(*
/*
 *****************************************************************************
 * timeUTCToJD: convert struct ccsTIMEVAL into Julian date
 *
 *  IN   ut: time in UT
 *  OUT    : Julian date  
 ***************************************************************************** 
 */
*)
FUNCTION F_timeUTCToJD : LREAL
VAR_INPUT
	ut:	T_TIMEVAL;
END_VAR
VAR
	temp1:	LREAL;
END_VAR

(*
DOUBLE timeUTCToJD(vltTIMEVAL *ut)    /* time in UT                       */
    {
    DOUBLE jd;
    
   /*
    * CONST4 = jd(70-01-01 00:00:00.000000)
    */
    jd = CONST4 + (ut->tv_sec + ut->tv_usec/1000000.)/86400.;
    return(jd);
    }
*)

//F_timeUTCToJD := GCL.C_CONST4 + (UDINT_TO_REAL(ut.tv_sec) + DINT_TO_REAL(ut.tv_usec)/1000000.0)/86400.0;

temp1	:= DINT_TO_LREAL(ut.tv_usec)/1000000.0;
temp1	:= temp1 + UDINT_TO_LREAL(ut.tv_sec);

F_timeUTCToJD := GCL.C_CONST4 + (temp1)/86400.0;

END_FUNCTION

(* stored: Version 1.1.0.1, ProductVersion 3.1.4024.10
   POU F_timeUTCToJD: Id {0fe20a4c-58af-45bf-a6b0-727ce9f434ea}, SpecialFunc None *)
